FUNCTION_BLOCK T_ContainsComponentCompareResultTrue EXTENDS T_UnitTestBase
VAR
END_VAR

TestFinished();

END_FUNCTION_BLOCK

(* stored: Version 1.1.0.1, ProductVersion 3.1.4024.12
   POU T_ContainsComponentCompareResultTrue: Id {e60208ed-9066-4494-9717-1e67b98003a8}, SpecialFunc None *)
